PROGRAM MAIN
VAR
END_VAR

END_PROGRAM

(* stored: Version 1.1.0.1
   POU MAIN: Id {64cf3e97-3804-4926-8187-b690cb96d9b0} *)
